FUNCTION "Pilz" : Void
VAR_TEMP
  Ret_Val_1 : Int;
  Ret_Val_2 : Int;
  Ret_Val_3 : Int;
  Ret_Val_4 : Int;
END_VAR
BEGIN
  // Původní jazyk: LAD
  // Zdroj XML: EXPORT/Program blocks/OP010/10_Device/27_Pilz/Pilz.xml
  // --- LAD/FBD → SCL (orientační převod, jen pro revizi) ---
  // Network 1
  // Network 2
  // --- Poznámky / omezení převodu ---
  // Síť obsahuje nepodporované prvky (ponecháno jen jako komentář): Move(2), Not(1)
END_FUNCTION
